VAR_GLOBAL
// TcHmi
	aDataGridStationConfig	: ARRAY [0..GVL_StationConfig.nMaxStationCount - 1] OF ST_DataGridStationConfig;
	anValveMaskListToRecipe	: ARRAY [0..GVL_StationConfig.nMaxStationCount - 1] OF ARRAY [0..GVL_leakTestConfig.nMaxTestSteps - 1] OF DWORD;
END_VAR

(* stored: Version 1.1.0.1
   GVL GVL_TcHmi: Id {e66e5bb2-e186-0a7a-1eb9-6daef8b222c0} *)
